PROGRAM modbus_mapping
VAR
	bop_power_meter_modbus_read : modbus_analog_read;
	prexfer_power_meter_modbus_read : modbus_analog_read;
	prodxfer_power_meter_modbus_read : modbus_analog_read;
	barge_power_meter_modbus_read : modbus_analog_read;
	acid_power_meter_modbus_read : modbus_analog_read;
	bped_main_power_meter_modbus_read : modbus_analog_read;
	bped_stack_power_meter_modbus_read : modbus_analog_read;
	nf1_power_meter_modbus_read : modbus_analog_read;
	ro_power_meter_modbus_read : modbus_analog_read;
	rocip_power_meter_modbus_read : modbus_analog_read;
	nf2_power_meter_modbus_read : modbus_analog_read;
END_VAR

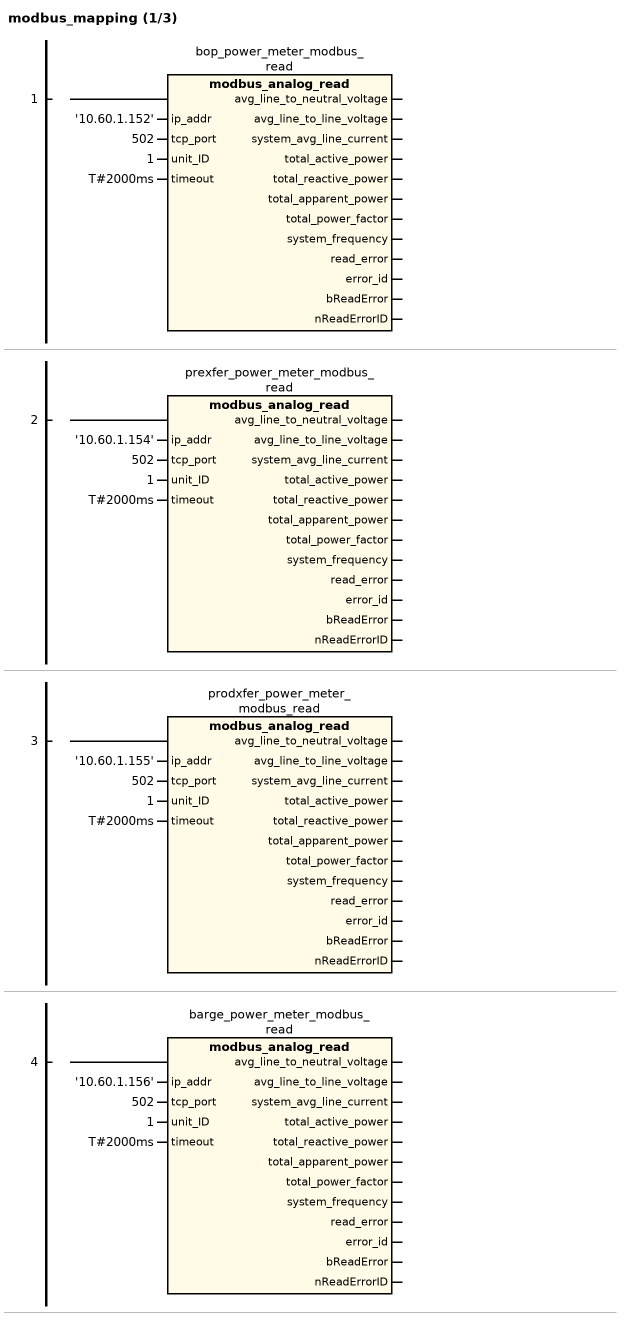
// NETWORK 1
bop_power_meter_modbus_read(ip_addr := '10.60.1.152', tcp_port := 502, unit_ID := 1, timeout := T#2000ms); // modbus_analog_read

// NETWORK 2
prexfer_power_meter_modbus_read(ip_addr := '10.60.1.154', tcp_port := 502, unit_ID := 1, timeout := T#2000ms); // modbus_analog_read

// NETWORK 3
prodxfer_power_meter_modbus_read(
    ip_addr := '10.60.1.155',
    tcp_port := 502,
    unit_ID := 1,
    timeout := T#2000ms); // modbus_analog_read

// NETWORK 4
barge_power_meter_modbus_read(ip_addr := '10.60.1.156', tcp_port := 502, unit_ID := 1, timeout := T#2000ms); // modbus_analog_read

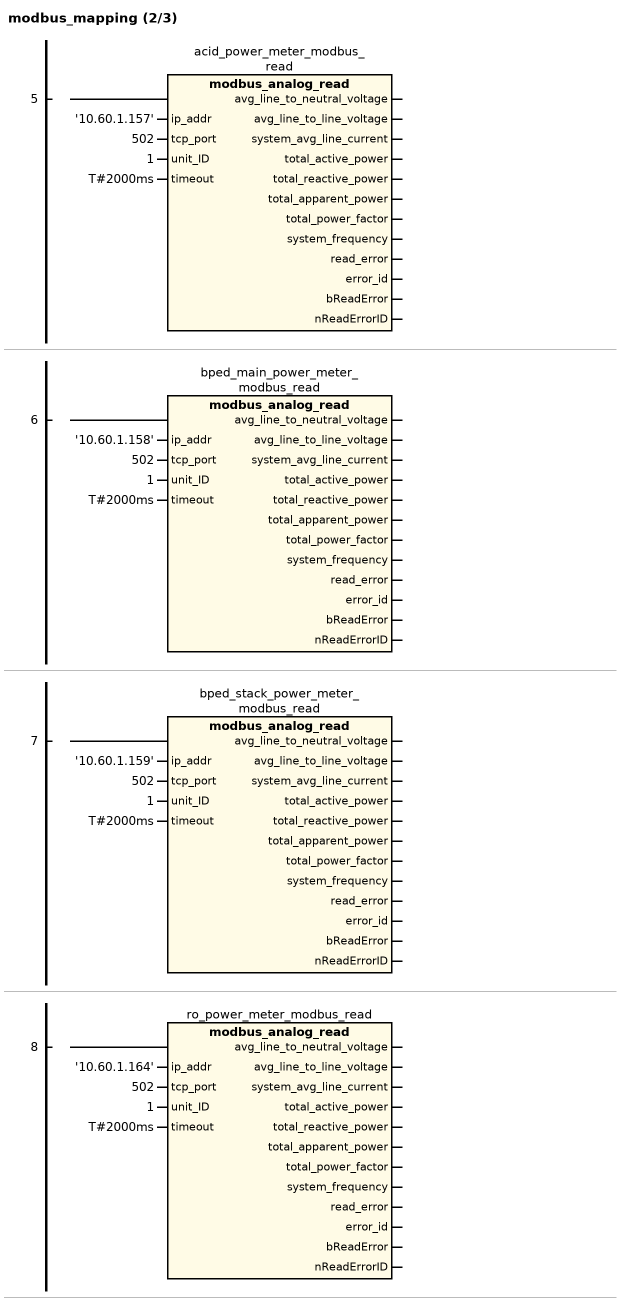
// NETWORK 5
acid_power_meter_modbus_read(ip_addr := '10.60.1.157', tcp_port := 502, unit_ID := 1, timeout := T#2000ms); // modbus_analog_read

// NETWORK 6
bped_main_power_meter_modbus_read(
    ip_addr := '10.60.1.158',
    tcp_port := 502,
    unit_ID := 1,
    timeout := T#2000ms); // modbus_analog_read

// NETWORK 7
bped_stack_power_meter_modbus_read(
    ip_addr := '10.60.1.159',
    tcp_port := 502,
    unit_ID := 1,
    timeout := T#2000ms); // modbus_analog_read

// NETWORK 8
ro_power_meter_modbus_read(ip_addr := '10.60.1.164', tcp_port := 502, unit_ID := 1, timeout := T#2000ms); // modbus_analog_read

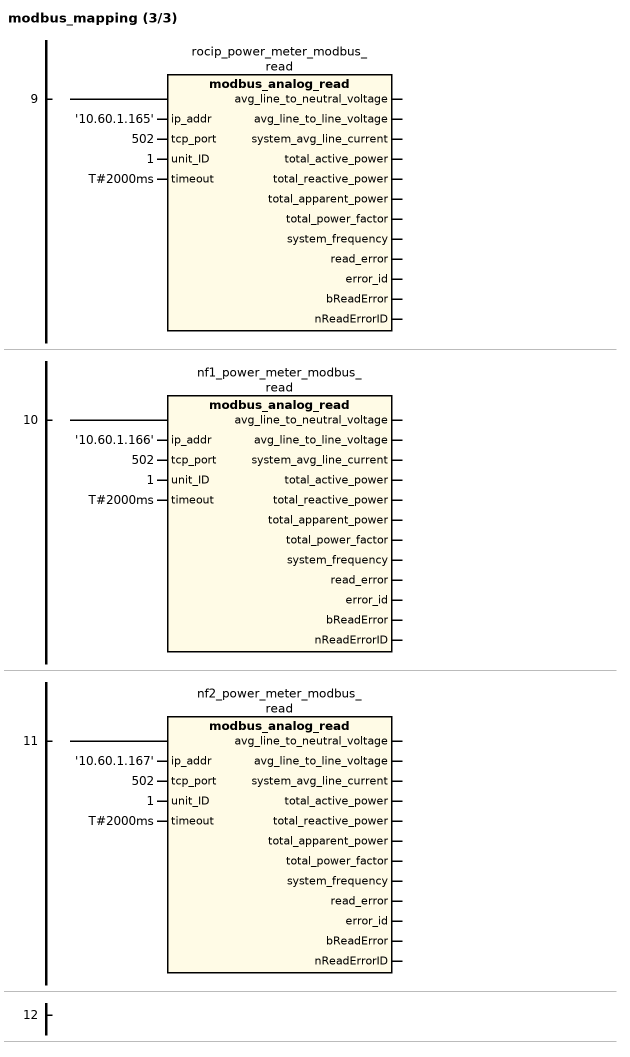
// NETWORK 9
rocip_power_meter_modbus_read(ip_addr := '10.60.1.165', tcp_port := 502, unit_ID := 1, timeout := T#2000ms); // modbus_analog_read

// NETWORK 10
nf1_power_meter_modbus_read(ip_addr := '10.60.1.166', tcp_port := 502, unit_ID := 1, timeout := T#2000ms); // modbus_analog_read

// NETWORK 11
nf2_power_meter_modbus_read(ip_addr := '10.60.1.167', tcp_port := 502, unit_ID := 1, timeout := T#2000ms); // modbus_analog_read

// NETWORK 12

END_PROGRAM

(* stored: Version 1.1.0.1, ProductVersion 3.1.4024.15
   POU modbus_mapping: Id {5fbe18e7-8052-475b-9627-0605698e2b4f}, SpecialFunc None *)
